FUNCTION F_LowestReal : REAL
VAR_INPUT
	Value1																: REAL;
	Value2																: REAL;
END_VAR
VAR
END_VAR

// F_LowerValue
// Rev 1.0 - March 14, 2024

F_LowestReal															:= SEL(Value1 < Value2, Value2, Value1);

END_FUNCTION

(* stored: Version 1.1.0.1, ProductVersion 3.1.4024.12
   POU F_LowestReal: Id {9e88cf8b-2020-4575-a920-4afa8023f33d}, SpecialFunc None *)
